PROGRAM FlowSequence_CC1Test
VAR_INPUT
	start : BOOL := FALSE;
	setSpeedDuration : TIME := T#15S;
	runTestDuration : TIME := T#2M;
	autoAdvance : BOOL := TRUE;
END_VAR
VAR_OUTPUT
	startTimes : ARRAY[1..50] OF ULINT;
	endTimes : ARRAY[1..50] OF ULINT;

	P9999Atubing : ARRAY[1..50] OF INT;
	P9999Btubing : ARRAY[1..50] OF INT;
END_VAR
VAR
	i : UINT := 0; // index
	n : UINT := 25;
	t : LREAL := 0.0;
	tol : LREAL := 5.0;
	spTotal : ARRAY [1..50] OF LREAL := [100.0,100.0,100.0,0.0,0.0,0.0,0.0,0.0,0.0,0.0,0.0,0.0,0.0,0.0,0.0,0.0,0.0,0.0,0.0,0.0,0.0,0.0,0.0,0.0, 0.0,
									0.0,0.0,0.0,0.0,0.0,0.0,0.0,0.0,0.0,0.0,0.0,0.0,0.0,0.0,0.0,0.0,0.0,0.0,0.0,0.0,0.0,0.0,0.0,0.0,0.0];
	//spTotal : ARRAY [1..50] OF LREAL := [100.0, 150.0, 200.0, 300.0, 150.0, 100.0, 80.0, 80.0, 90.0, 100.0, 
    //                                110.0, 120.0, 130.0, 140.0, 150.0, 0.0, 0.0, 0.0,
    //                                0.0, 0.0, 0.0, 0.0, 0.0, 0.0,
	//								0.0,0.0,0.0,0.0,0.0,0.0,0.0,0.0,0.0,0.0,0.0,0.0,0.0,0.0,0.0,0.0,0.0,0.0,0.0,0.0,0.0,0.0,0.0,0.0];
	spConc : ARRAY [1..50] OF LREAL := [1.0, 1.0, 1.0, 1.0, 1.0, 1.0, 1.0, 1.0, 1.0, 1.0, 
                                    1.0, 1.0, 1.0, 1.0, 1.0, 0.0, 0.0, 0.0,
                                    0.0, 0.0, 0.0, 0.0, 0.0, 0.0,
									0.0,0.0,0.0,0.0,0.0,0.0,0.0,0.0,0.0,0.0,0.0,0.0,0.0,0.0,0.0,0.0,0.0,0.0,0.0,0.0,0.0,0.0,0.0,0.0];
	
	setSpeed : SFCStepType;
	runTest : SFCStepType;
	recordTest : SFCStepType;
END_VAR

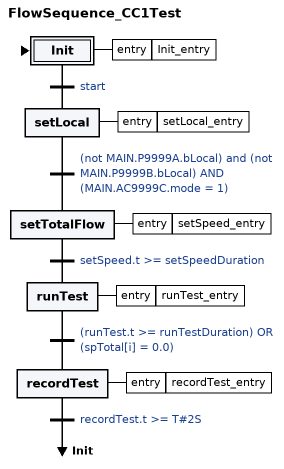
INITIAL_STEP Init:
    Init_entry(P1);  // entry action
END_STEP
TRANSITION FROM Init TO setLocal
    := start;
END_TRANSITION
STEP setLocal:
    setLocal_entry(P1);  // entry action
END_STEP
TRANSITION FROM setLocal TO setTotalFlow
    := (not MAIN.P9999A.bLocal) and (not MAIN.P9999B.bLocal) AND (MAIN.AC9999C.mode = 1);
END_TRANSITION
STEP setTotalFlow:
    setSpeed_entry(P1);  // entry action
END_STEP
TRANSITION FROM setTotalFlow TO runTest
    := setSpeed.t >= setSpeedDuration;
END_TRANSITION
STEP runTest:
    runTest_entry(P1);  // entry action
END_STEP
TRANSITION FROM runTest TO recordTest
    := (runTest.t >= runTestDuration) OR (spTotal[i] = 0.0);
END_TRANSITION
STEP recordTest:
    recordTest_entry(P1);  // entry action
END_STEP
TRANSITION FROM recordTest TO Init
    := recordTest.t >= T#2S;
END_TRANSITION

ACTION setLocal_entry:
IF MAIN.P9999A.bLocal THEN
	MAIN.P9999A.nLocal_RQ := 0;  //put pump in remote
END_IF
IF MAIN.P9999B.bLocal THEN
	MAIN.P9999B.nLocal_RQ := 0;  //put pump in remote
END_IF

IF MAIN.AC9999C.mode <> 1 THEN // concentration control in auto
	MAIN.AC9999C.c.rq := 0; // set initial total flow
	MAIN.AC9999C.conc.rq := 1.0; // set initial concentration
	MAIN.AC9999C.mode := 1;
END_IF
END_ACTION

ACTION Init_entry:
IF i >= n THEN
	MAIN.AC9999C.mode := 0; // concentration control in manual
	MAIN.P9999A.nRun_RQ := 0; //stop pump
	MAIN.P9999B.nRun_RQ := 0; //stop pump
	start := FALSE;
	i := 0;
END_IF
MAIN.logActive := FALSE;
END_ACTION

ACTION resetTotals_entry:
MAIN.fbFQ9999A.resetRQ := TRUE;
MAIN.fbFQ9999B.resetRQ := TRUE;
MAIN.fbFQ9999C.resetRQ := TRUE;
MAIN.MTSendString := 'ZI$0D$0A';
MAIN.logActive := TRUE;
END_ACTION

ACTION runTest_entry:
MAIN.MTSendString := 'SIR$0D$0A';
startTimes[i] := unixTime;
END_ACTION

ACTION setSpeed_entry:
i := i + 1;
startTimes[i] := 0;
endTimes[i] := 0;

MAIN.AC9999C.c.rq := spTotal[i];
MAIN.AC9999C.conc.rq := spConc[i];

P9999Atubing[i] := MAIN.P9999A.nTubeSize;
P9999Btubing[i] := MAIN.P9999B.nTubeSize;
END_ACTION

ACTION recordTest_entry:
endTimes[i] := unixTime;

t := DWORD_TO_LREAL(TIME_TO_DWORD(runTestDuration))/1000.0/60.0;

IF NOT autoAdvance THEN
	start := FALSE;
END_IF
END_ACTION

END_PROGRAM

(* stored: Version 1.1.0.1, ProductVersion 3.1.0.36
   POU FlowSequence_CC1Test: Id {bf733076-098a-4137-a94d-1dac27d2645f}, SpecialFunc None
   Action setLocal_entry: Id {013f24c3-125a-4c91-a319-ad21f2ec3071}
   Action Init_entry: Id {2f9dcdd8-ea44-4f9e-92f5-f4d1c2243fdc}
   Action resetTotals_entry: Id {48990d29-8a8c-44f0-8e7b-53c307d47b6e}
   Action runTest_entry: Id {800ca229-8577-4e86-bc02-9831bbb33a52}
   Action setSpeed_entry: Id {df37f69c-63b3-45e3-959a-cb61b1ced2c8}
   Action recordTest_entry: Id {ef9d28c0-abd7-46b6-a0b9-356a08629c77} *)
